// Code généré automatiquement : NE PAS MODIFIER
FUNCTION CheckRangeUnsigned : UDINT
VAR_INPUT
	value, lower, upper: UDINT;
END_VAR

// Code généré automatiquement : Il s’agit d’une proposition d’implémentation.
{noflow}
IF (value < lower) THEN
	CheckRangeUnsigned := lower;
ELSIF(value > upper) THEN
	CheckRangeUnsigned := upper;
ELSE
	CheckRangeUnsigned := value;
END_IF
{flow}

END_FUNCTION

(* stored: Version 1.1.0.1, ProductVersion 3.1.4024.6
   POU CheckRangeUnsigned: Id {ae628837-05cc-4aad-9c35-cc6645c0a6a9}, SpecialFunc CheckRangeUnsigned *)
